Staubli VAL3: onStart.pgx

program onStart(num x_nResult)
  local bool l_bOk
  local string l_sButton[2]
  local string l_sMessage
  local string l_sPage
  local string l_sItem
begin
  // clean the movement
  if !isEmpty()
    resetMotion()
  endIf
  nPoint=0
  cls()
  bStepping=false
  // save the traj Name
  sTrajName=sItems
  // INIT the resource
  use:bUseRefresh=true
  // load all
  call loadType(x_nResult)
  //
  // look if the trajType has the stepping enable
  //
  if trajType:bStepping
    call loadEditTraj(sTrajName)
    //
    logMsg("[KERNEL] INTERFACE:PAGE Simulation")
  else
    // only start and return
    call language:message(l_sMessage,214)
    call language:getYesNo(l_sButton)
    // ask the yes_no question
    call use:yes_no(l_sMessage,l_sButton,l_bOk)
    if l_bOk
      cycleStatus:iToSuperV.sType=saveData:sTrajTypeUsing
      cycleStatus:iToSuperV.sData=sTrajName
      cycleStatus:nInterfaceToSV=3
      logMsg("[KERNEL] INTERFACE:Simulation of the item: "+saveData:sTrajTypeUsing+" "+sTrajName)
      wait(cycleStatus:nInterfaceToSV==-1)
      // load the production page
      l_sPage="kernel/page/production"
      l_sItem="simulation"
      call loadPage(l_sPage,l_sItem)
      call use:setView(false)
    endIf
    x_nResult=99
  endIf
  //
end
